// TIA Portal V20 export
FUNCTION_BLOCK "FB_GestionFixture"   // FB49, SCL
{ S7_Optimized_Access := 'TRUE' }
// stored: MemoryReserve 100, SetENOAutomatically false
   VAR RETAIN
      sFixtureHold : Bool;
   END_VAR
   VAR
      sFixtureVacuum : Bool;
      sFixtureBlowing : Bool;
      sFixtureStandard { S7_SetPoint := 'True'} : "FB_Fixture";
      sFixtureStandardErrorCode { S7_SetPoint := 'True'} : Int;
      sFixturePartControl : "FB_PartPresenceCtrl";
      sRT_VacuumStartReq { S7_SetPoint := 'True'} : R_TRIG;
      sRT_VacuumStopReq { S7_SetPoint := 'True'} : R_TRIG;
   END_VAR
   VAR_TEMP
      tFixtureOpenAllowed : Bool;
      tFixtureCloseAllowed : Bool;
      tNull : Bool;
   END_VAR
   VAR CONSTANT
      B_AXIS_POSITION_MIN : Real := 0.0;   // B Axis Pos. Min to allow fixture opening
      B_AXIS_POSITION_MAX : Real := 15.0;   // B Axis Pos. Max to allow fixture opening
      V_AXIS_POSITION_MIN : Real := -1.0;   // V Axis Pos. Min to allow fixture opening/closing
      V_AXIS_POSITION_MAX : Real := 15.0;   // V Axis Pos. Max to allow fixture opening/closing
      W_AXIS_POSITION_MIN : Real := 0.0;   // W Axis Pos. Min to allow fixture opening/closing
      W_AXIS_POSITION_MAX : Real := 15.0;   // W Axis Pos. Max to allow fixture opening/closing
   END_VAR
BEGIN
   REGION Description header 
       //==================================================================================
       // POSALUX Swiss SA / (C) Copyright 2025
       //----------------------------------------------------------------------------------
       // Title: Structure sequence
       // Comment/Function: 
       //
       // Author: Fabien Waldt
       // Engineering: TIA Portal v17
       //----------------------------------------------------------------------------------
       // Change log table:
       // Version  | Date     | Expert in charge | Changes applied
       // ---------|----------|------------------|------------------------------------
       // 00.00.01 | 20250219 | WFA              | First released version
       // ==================================================================================
   END_REGION

   REGION
       #tFixtureOpenAllowed := ("DB_AxisPosition".sAxis04_B."$AA_IM" >= #B_AXIS_POSITION_MIN  AND "DB_AxisPosition".sAxis04_B."$AA_IM" <= #B_AXIS_POSITION_MAX)
                           AND ("DB_AxisPosition".sAxis07_V."$AA_IM" >= #V_AXIS_POSITION_MIN  AND "DB_AxisPosition".sAxis08_W."$AA_IM" >= #W_AXIS_POSITION_MIN);
       #tFixtureCloseAllowed := ("DB_AxisPosition".sAxis07_V."$AA_IM" >= #V_AXIS_POSITION_MIN AND "DB_AxisPosition".sAxis08_W."$AA_IM" >= #W_AXIS_POSITION_MIN);
   END_REGION

   REGION HOLD CLAMP
       REGION F_Hold Key Disable + channel switch Key[7]
       // Hold Key[7] disable 
           "DB_McpKeyboardSignals".sK7_FixtureClamp.sKeyDisable := "LBP_Chan1".E_ProgRunning OR "DB_GestionWorkingModes".sMCP_KxxKeysDisable;
            "DB_HmiKeyboardSignals".sK7_FixtureClamp.sKeyDisable := "LBP_Chan1".E_ProgRunning;
       // Force toggle Key[7] when hold is active    
            "DB_McpKeyboardSignals".sK7_FixtureClamp.sKeySWToggleStatus := #sFixtureHold;
            "DB_HmiKeyboardSignals".sK7_FixtureClamp.sKeySWToggleStatus := #sFixtureHold;
   END_REGION

   REGION Fixture 1 
       REGION Clamping Management
           // Hold signal for clamping - M84: Hold clamp
           IF #tFixtureCloseAllowed THEN
               IF "LBP_Chan1".MDyn[84]                                 // M84: Hold clamp
                   OR "DB_McpKeyboardSignals".sK7_FixtureClamp.sKeySWTogglePositiveFront
                   OR "DB_HmiKeyboardSignals".sK7_FixtureClamp.sKeySWTogglePositiveFront
                   OR "LBP_ModeGroup".A_REF
                   OR "DB_LoaderFixture".oFixtureCloseReq THEN
                   #sFixtureHold := TRUE;
                   "DB_McpKeyboardSignals".sK7_FixtureClamp.sKeySWToggleStatus := TRUE;
                   "DB_HmiKeyboardSignals".sK7_FixtureClamp.sKeySWToggleStatus := TRUE;
               END_IF;
           END_IF;
           // Release signal for clamping - M85: Release clamp
           IF #tFixtureOpenAllowed THEN
               IF "LBP_Chan1".MDyn[85]                                 // M85: Release clamp
                   OR "DB_McpKeyboardSignals".sK7_FixtureClamp.sKeySWToggleNegativeFront
                   OR "DB_HmiKeyboardSignals".sK7_FixtureClamp.sKeySWToggleNegativeFront
                   OR "DB_LoaderFixture".oFixtureOpenReq THEN
                   #sFixtureHold := FALSE;
                   "DB_McpKeyboardSignals".sK7_FixtureClamp.sKeySWToggleStatus := FALSE;
                   "DB_HmiKeyboardSignals".sK7_FixtureClamp.sKeySWToggleStatus := FALSE;
               END_IF;
           END_IF;
       END_REGION
   END_REGION
   END_REGION

   REGION F_Hold LED[7]
       "DB_McpKeyboardSignals".sK7_FixtureClamp.sLedSWStatus := #sFixtureHold;
       "DB_HmiKeyboardSignals".sK7_FixtureClamp.sLedSWStatus := #sFixtureHold;
   END_REGION

   REGION VACUUM
       REGION F_Vacuum Key Disable + Channel switch Key[8]
           // Vacuum Key[8] disable
           "DB_McpKeyboardSignals".sK8_FixtureVacuum.sKeyDisable := "LBP_Chan1".E_ProgRunning OR "DB_GestionWorkingModes".sMCP_KxxKeysDisable;
           "DB_HmiKeyboardSignals".sK8_FixtureVacuum.sKeyDisable := "LBP_Chan1".E_ProgRunning;

           // Force TOGGLE Key[8] when Vacuum is active    
           "DB_McpKeyboardSignals".sK8_FixtureVacuum.sKeySWToggleStatus := #sFixtureVacuum;
           "DB_HmiKeyboardSignals".sK8_FixtureVacuum.sKeySWToggleStatus := #sFixtureVacuum;
       END_REGION

       REGION Fixture 1
           #sRT_VacuumStartReq(CLK := "DB_LoaderFixture".sFixtureLoading.oVacuumStartReq);
           #sRT_VacuumStopReq(CLK := "DB_LoaderFixture".sFixtureUnloading.oVacuumStopReq);

           // Fixture Vacuum ON - M86: Vacuum ON
           IF "LBP_Chan1".MDyn[86]
               OR #sRT_VacuumStartReq.Q
               OR "DB_McpKeyboardSignals".sK8_FixtureVacuum.sKeySWTogglePositiveFront 
               OR "DB_HmiKeyboardSignals".sK8_FixtureVacuum.sKeySWTogglePositiveFront THEN
                   #sFixtureVacuum := TRUE;
                   "DB_McpKeyboardSignals".sK8_FixtureVacuum.sKeySWToggleStatus := TRUE;
                   "DB_HmiKeyboardSignals".sK8_FixtureVacuum.sKeySWToggleStatus := TRUE;
           END_IF;

           // Fixture Vacuum OFF (Station 1) - M87: Vacuum OFF
           IF "LBP_Chan1".MDyn[87]
               OR #sRT_VacuumStopReq.Q
               OR "DB_McpKeyboardSignals".sK8_FixtureVacuum.sKeySWToggleNegativeFront 
               OR "DB_HmiKeyboardSignals".sK8_FixtureVacuum.sKeySWToggleNegativeFront THEN
                   #sFixtureVacuum := FALSE;
                   "DB_McpKeyboardSignals".sK8_FixtureVacuum.sKeySWToggleStatus := FALSE;
                   "DB_HmiKeyboardSignals".sK8_FixtureVacuum.sKeySWToggleStatus := FALSE;
           END_IF;
       END_REGION

       REGION F_Vacuum LED[8]
           "DB_McpKeyboardSignals".sK8_FixtureVacuum.sLedSWStatus := #sFixtureVacuum;
           "DB_HmiKeyboardSignals".sK8_FixtureVacuum.sLedSWStatus := #sFixtureVacuum;
       END_REGION
   END_REGION

   REGION Standard Fixture
       #sFixtureStandard(iOpenCtrl := "DB_DigitalInputs".sClampingOpenCtrl.sSWStatus,
                         iCloseCtrl :="DB_DigitalOutputs".sClampingClosing.sSWStatus,
                         iHoldReq := #sFixtureHold,
                         iVacuumReq := #sFixtureVacuum,
                         iBlowingReq := #sFixtureBlowing,
                         iMonitorTime := T#2s,
                         oClampOpening => "DB_DigitalOutputs".sClampingOpening.sSWStatus,
                         oClampClosing => "DB_DigitalOutputs".sClampingClosing.sSWStatus,
                         oVacuumActivation => "DB_DigitalOutputs".sSuction.sSWStatus,
                         oBlowingActivation => #tNull, // No Blowing
                         oErrorCode => #sFixtureStandardErrorCode);
   END_REGION

   REGION Station 1 Fixture Alarms
       "LBP_AlarmMsgs".UserA[08].A70UUxx[12] := #sFixtureStandardErrorCode = 1;    // Msg: 700812 "Fixture Opening Timeout"
       "LBP_AlarmMsgs".UserA[08].A70UUxx[13] := #sFixtureStandardErrorCode = 2;    // Msg: 700813 "Fixture Closing Timeout"
   END_REGION

   REGION Fixture Part Control
       // Measure > iProdOK_LimHigh                          => Bad Positionning
       // iProdOK_LimLow <= Measure <= iProdOK_LimHigh       => Good part
       // NOT (iProdOK_LimLow <= Measure <= iProdOK_LimHigh) => Bad part
       // iProdMissing <= Measure <= iProdOK_LimLow          => Missing Backwall   (NOT POSSIBLE FOR FL.0153)
       // Measure < iProdMissing                             => Missing Part       (NOT POSSIBLE FOR FL.0153)
       // Teach-in :
           // ProdOK_LimHigh
           // ProdOK_LimLow
           // ProdMissing  (NOT USED FOR FL.0153)

       #sFixturePartControl.iProdOK_LimHigh := 25000; // WFA A supprimer quand recette OK
       #sFixturePartControl.iProdOK_LimLow := 9500; // WFA A supprimer quand recette OK
       // Voir dans FB_Recipe les transferts des limites High et Low

       #sFixturePartControl("iStart Control" := ("DB_LoaderFixture".oFixtureCloseReq OR "DB_DigitalOutputs".sClampingClosing.sSWStatus),             // M84: Hold clamp
                            iMeasureValue := "DB_AnalogInputs".sAxisB_ClampingPart.sSWRealValue,
                            iProdOK_LimHigh := #sFixturePartControl.iProdOK_LimHigh,
                            iProdOK_LimLow := #sFixturePartControl.iProdOK_LimLow,
                            iProdMissing:= #sFixturePartControl.iProdMissing,
                            oGoodPart => #sFixturePartControl.oGoodPart,
                            oBadpart => #sFixturePartControl.oBadpart);
   END_REGION

    REGION RID Fixture mvt
         "LBP_AlarmMsgs".Chan[1].RID[10] := #sFixtureStandard.oClampClosing AND NOT #sFixtureStandard.iCloseCtrl
         OR #sFixtureStandard.oClampOpening AND NOT #sFixtureStandard.iOpenCtrl;
    END_REGION
END_FUNCTION_BLOCK
